FUNCTION BYTE_TO_SIZE : ST_SIZE
VAR_INPUT
	nValue : BYTE;
END_VAR

BYTE_TO_SIZE.nValue := nValue;

END_FUNCTION

(* stored: Version 1.1.0.1, ProductVersion 3.1.4024.15
   POU BYTE_TO_SIZE: Id {b4ddb272-de98-4c80-8b4d-11faba84d6a1}, SpecialFunc None *)
